// TIA Portal V16 export
// export: Created 2019-09-22T13:16:38.3602951Z, ExportSetting WithDefaults, DisplayName Totally Integrated Automation Portal, DisplayVersion V16, DisplayName TIA Portal Version Control Interface, DisplayVersion V16, DisplayName TIA Portal Openness, DisplayVersion V16, DisplayName STEP 7 Professional, DisplayVersion V16, DisplayName SIMATIC Energy Suite, DisplayVersion V16, DisplayName STEP 7 Safety, DisplayVersion V16, DisplayName WinCC Professional, DisplayVersion V16, DisplayName SIMATIC Visualization Architect, DisplayVersion V16
FUNCTION_BLOCK "MainFB"   // FB200, FBD
{ S7_Optimized_Access := 'TRUE' }
VERSION : 0.1
// stored: AutoNumber true, IsIECCheckEnabled false, IsRetainMemResEnabled false, MemoryReserve 100, SetENOAutomatically false, UDAEnableTagReadback false
   VAR_INPUT
      initialCall { ExternalAccessible := 'False'; ExternalVisible := 'False'; ExternalWritable := 'False'} : Bool;   // Initial call of this OB
   END_VAR
   VAR
      instLiftStartStop { S7_SetPoint := 'True'} : "LiftStartStop";
      instLift1Cmd { S7_SetPoint := 'True'} : "LiftCmd";
      instLift2Cmd { S7_SetPoint := 'True'} : "LiftCmd";
   END_VAR
BEGIN

REGION Network 1: common
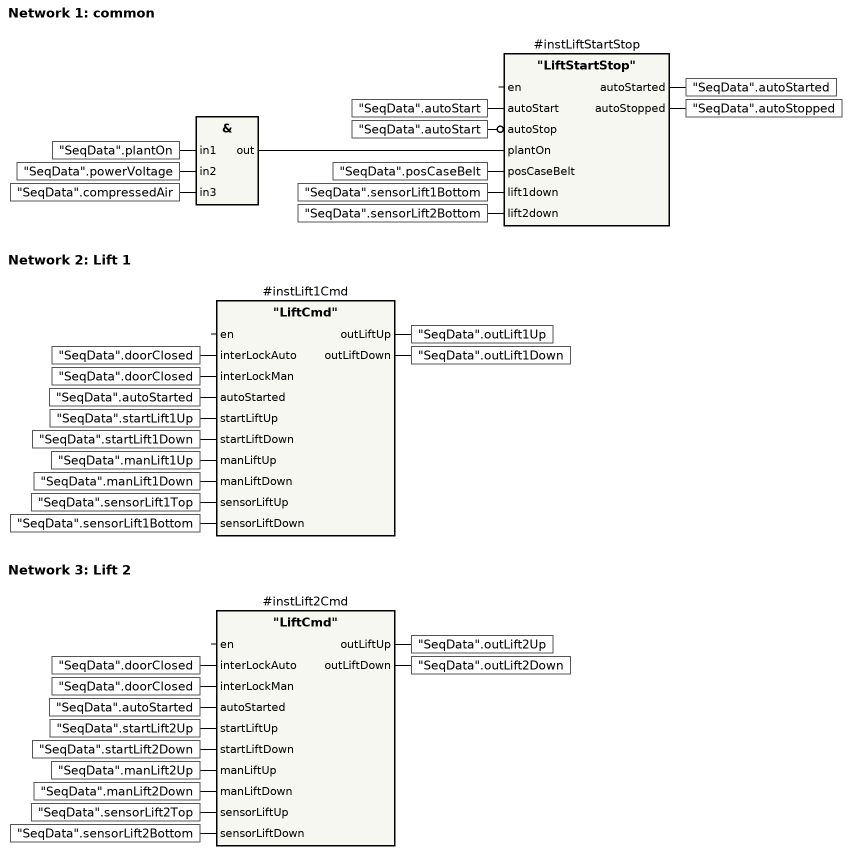
   #instLiftStartStop(autoStart := "SeqData".autoStart,   // "LiftStartStop"
                      autoStop := NOT "SeqData".autoStart,
                      plantOn := "SeqData".plantOn AND "SeqData".powerVoltage AND "SeqData".compressedAir,
                      posCaseBelt := "SeqData".posCaseBelt,
                      lift1down := "SeqData".sensorLift1Bottom,
                      lift2down := "SeqData".sensorLift2Bottom,
                      autoStarted => "SeqData".autoStarted,
                      autoStopped => "SeqData".autoStopped);
END_REGION

REGION Network 2: Lift 1
   #instLift1Cmd(interLockAuto := "SeqData".doorClosed,   // "LiftCmd"
                 interLockMan := "SeqData".doorClosed,
                 autoStarted := "SeqData".autoStarted,
                 startLiftUp := "SeqData".startLift1Up,
                 startLiftDown := "SeqData".startLift1Down,
                 manLiftUp := "SeqData".manLift1Up,
                 manLiftDown := "SeqData".manLift1Down,
                 sensorLiftUp := "SeqData".sensorLift1Top,
                 sensorLiftDown := "SeqData".sensorLift1Bottom,
                 outLiftUp => "SeqData".outLift1Up,
                 outLiftDown => "SeqData".outLift1Down);
END_REGION

REGION Network 3: Lift 2
   #instLift2Cmd(interLockAuto := "SeqData".doorClosed,   // "LiftCmd"
                 interLockMan := "SeqData".doorClosed,
                 autoStarted := "SeqData".autoStarted,
                 startLiftUp := "SeqData".startLift2Up,
                 startLiftDown := "SeqData".startLift2Down,
                 manLiftUp := "SeqData".manLift2Up,
                 manLiftDown := "SeqData".manLift2Down,
                 sensorLiftUp := "SeqData".sensorLift2Top,
                 sensorLiftDown := "SeqData".sensorLift2Bottom,
                 outLiftUp => "SeqData".outLift2Up,
                 outLiftDown => "SeqData".outLift2Down);
END_REGION
END_FUNCTION_BLOCK
